{attribute 'GeneratedUsingTerminal: EPP6001-0002-0016'}
{attribute addProperty BoxType "EPP6001-0002-0016"}
{attribute addProperty Id "COM_InputsAT %I*COM_Inputs_6C2FC20224COM_OutputsAT %Q*COM_Outputs_5D00B5E724WcStateAT %I*WcState_9091E0EB2InfoDataAT %I*InfoData_32EB74EA10"}
{attribute addProperty CRC "1082670339"}
{attribute addProperty Size "60"}
TYPE EPP6001_40883D03 EXTENDS EtcSlaveTerminalBase_947E5A46 :
STRUCT
	{attribute addProperty Name "COM_Inputs"}
	COM_Inputs : COM_Inputs_6C2FC202;
	{attribute addProperty Name "COM_Outputs"}
	COM_Outputs : COM_Outputs_5D00B5E7;
	{attribute addProperty Name "WcState"}
	WcState : WcState_9091E0EB;
	{attribute addProperty Name "InfoData"}
	InfoData : InfoData_32EB74EA;
END_STRUCT
END_TYPE

(* stored: Version 1.2.0.0, ProductVersion 3.1.4024.9
   DUT EPP6001_40883D03: Id {80aac684-64da-44f9-a075-86a69397e615} *)
